Staubli VAL3: onF1Event.pgx

program onF1Event()
  local num l_nJogVelocity
  local num l_nSpeedScale
begin
  // look if the bButton is enable
  if bButton[0]
    // decrease the move


    ////    io:direction_neg=true
    ////    wait(getKey()==-1)
    ////    io:direction_neg=false




    if aioGet(MbAI_b8MotorPow)==1
      //8轴移动速度

      l_nJogVelocity=2
      /////
      aioSet(MbAO_aJogVelo8,l_nJogVelocity)
      aioSet(MbAO_bMoveDirM,1)
      aioSet(MbAO_b8Axis,1)
      call use:timerDialog("8轴负向移动...",0)
    else
      if aioGet(MbAI_b8MotorPow)==0
        call use:timerDialog("8轴未上电",1)
        return
      endIf
    endIf


  endIf
  //

end
